(* Logix 5000 project; controller ktc_exapmple2 vendor 1 type 14 code 150 rev 30.11; software revision 30.00 *)

TASK MainTask (continuous, watchdog 500 ms) : MainProgram

MODULES
   Local : vendor 1 type 14 code 150 (Compact 0, rev 30.11)
      Counters : Embedded (Compact 3, rev 1.1, Output RPI 20 ms)
      Discrete_IO : Embedded (Compact 1, rev 3.1, Output RPI 20 ms)
      Analog_IO : Embedded (Compact 2, rev 1.1, Output RPI 80 ms)
END_MODULES

PROGRAM MainProgram   (* main routine MainRoutine *)
VAR
   LED_1 : BOOL;
   PB_1 : ALIAS FOR Local:1:I.Data.1;   // PUSH BUTTON NO
   PB_2 : ALIAS FOR Local:1:I.Data.0;   // PUSH BUTTON NO
   PL_1 : ALIAS FOR Local:1:O.Data.7;   // LED 7
   PL_2 : ALIAS FOR Local:1:O.Data.1;   // LED1
   PL_3 : ALIAS FOR Local:1:O.Data.2;   // LED 3
   PL_4 : ALIAS FOR Local:1:O.Data.6;   // LED 6
   SW_1 : ALIAS FOR Local:1:I.Data.6;   // SWITCH
END_VAR

ROUTINE MainRoutine   (* ladder *)
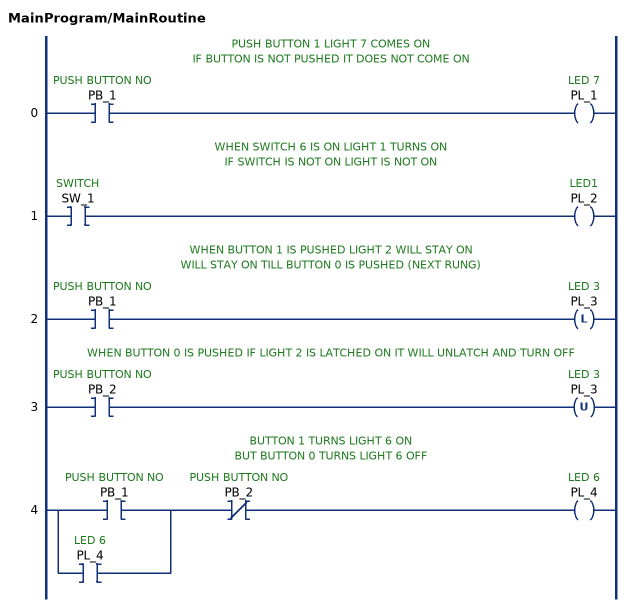
   // PUSH BUTTON 1 LIGHT 7 COMES ON
   // IF BUTTON IS NOT PUSHED IT DOES NOT COME ON
   0: XIC(PB_1)OTE(PL_1);
   // WHEN SWITCH 6 IS ON LIGHT 1 TURNS ON
   // IF SWITCH IS NOT ON LIGHT IS NOT ON
   1: XIC(SW_1)OTE(PL_2);
   // WHEN BUTTON 1 IS PUSHED LIGHT 2 WILL STAY ON
   // WILL STAY ON TILL BUTTON 0 IS PUSHED (NEXT RUNG)
   2: XIC(PB_1)OTL(PL_3);
   // WHEN BUTTON 0 IS PUSHED IF LIGHT 2 IS LATCHED ON IT WILL UNLATCH AND TURN OFF
   3: XIC(PB_2)OTU(PL_3);
   // BUTTON 1 TURNS LIGHT 6 ON
   // BUT BUTTON 0 TURNS LIGHT 6 OFF
   4: [XIC(PB_1) ,XIC(PL_4) ]XIO(PB_2)OTE(PL_4);
END_ROUTINE
END_PROGRAM
